FUNCTION_BLOCK MultipleEMerge (* Basic Function Block Type *)
  (* Standard: 61499-2 *)
  (* Version 0.0, 11/1/2016, chivdan, nxtControl GmbH, Template *)
  PACKAGE Main;
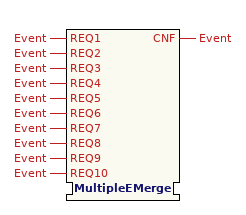
  EVENT_INPUT
    REQ1; (* Normal Execution Request *)
    REQ2;
    REQ3;
    REQ4;
    REQ5;
    REQ6;
    REQ7;
    REQ8;
    REQ9;
    REQ10;
  END_EVENT
  EVENT_OUTPUT
    CNF; (* Execution Confirmation *)
  END_EVENT
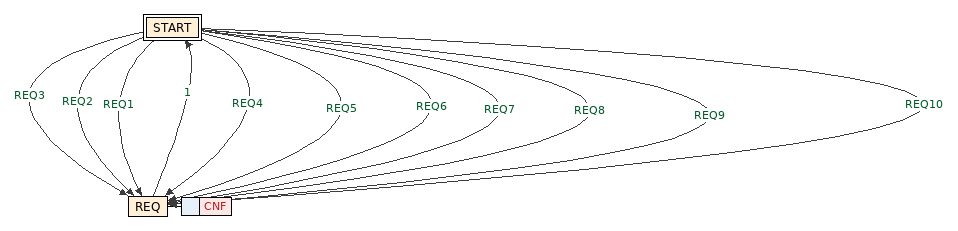
  EC_STATES
    START; (* Initial State *)
    REQ : -> CNF; (* Normal execution *)
  END_STATES
  EC_TRANSITIONS
    START TO REQ := REQ1;
    REQ TO START := 1;
    START TO REQ := REQ2;
    START TO REQ := REQ3;
    START TO REQ := REQ4;
    START TO REQ := REQ5;
    START TO REQ := REQ6;
    START TO REQ := REQ7;
    START TO REQ := REQ8;
    START TO REQ := REQ9;
    START TO REQ := REQ10;
  END_TRANSITIONS
END_FUNCTION_BLOCK
